FUNCTION_BLOCK FB_MotionDevices EXTENDS FB_HMIBase
VAR
	binary : Discrete.I_DiscreteBase;
END_VAR

METHOD Cyclic
VAR
END_VAR
// Sync status from device to HMI
status.HmiStatus.Busy := binary.P_DiscreteStatus.ComponentStatus.BaseStatus.Busy;
status.HmiStatus.Done := binary.P_DiscreteStatus.ComponentStatus.BaseStatus.Done;
status.HmiStatus.Error := binary.P_DiscreteStatus.ComponentStatus.BaseStatus.Error;

// Map discrete state to Enabled flag
status.HmiStatus.Enabled := (binary.P_DiscreteStatus.BinaryComponentState = Discrete.E_DiscreteComponentState.Active);

// Handle commands from Vue.js
IF cmd.Enable THEN
	binary.Activate();
	cmd.Enable := FALSE;
END_IF

IF cmd.Disable THEN
	binary.Deactivate();
	cmd.Disable := FALSE;
END_IF
END_METHOD

METHOD Init : BOOL
VAR_INPUT
	refBinary : Discrete.I_DiscreteBase;
END_VAR
binary := refBinary;
Init := TRUE;
END_METHOD

END_FUNCTION_BLOCK

(* stored: Version 1.1.0.1
   POU FB_MotionDevices: Id {6561488d-5d31-48fa-9698-23146b5d0312}, SpecialFunc None
   Method Cyclic: Id {b41161a6-18ca-4275-b0ae-52d268e55440}
   Method Init: Id {e266e6fc-c9f6-411e-9941-87a945869314} *)
